FUNCTION_BLOCK FB_Parent
VAR_INPUT
END_VAR
VAR_OUTPUT
END_VAR
VAR
	ref_child : REFERENCE TO FB_Child;
	m_parent_data : ARRAY [0..1023] OF REAL;
END_VAR

END_FUNCTION_BLOCK

(* stored: Version 1.1.0.1, ProductVersion 3.1.4024.12
   POU FB_Parent: Id {291b6a94-190c-4903-85c0-ad087a0adcde}, SpecialFunc None *)
